{attribute wpf [Container(Layout.Stack)]}
FUNCTION_BLOCK TcoKeyNormalService EXTENDS TcoElements.TcoDi IMPLEMENTS ITcoKeyNormalSevice

VAR

	
	{attribute addProperty Name "<#Key state#> - <#Service#>"}
	_isKeyInService           : BOOL; 

	{attribute addProperty Name "<#Key state#> - <#Normal#>"}
	_isKeyInNormal            : BOOL; 
END_VAR

SUPER^(inoSignal:= inoSignal);


THIS^._isKeyInNormal :=NOT THIS^._signal ;
THIS^._isKeyInService := NOT THIS^._isKeyInNormal;

PROPERTY KeyInNormal : BOOL
GET
KeyInNormal := _isKeyInNormal;
END_GET
END_PROPERTY

PROPERTY KeyInService : BOOL
GET
KeyInService := _isKeyInService;
END_GET
END_PROPERTY

END_FUNCTION_BLOCK

(* stored: Version 1.1.0.1
   POU TcoKeyNormalService: Id {fd8dbc27-6e45-4e78-8f75-e78a5510e99d}, SpecialFunc None
   Property KeyInNormal: Id {ec1426ec-5fce-4c25-9228-d7d73b4c1d65}
   Get Get: Id {0831bc1d-0f68-4b95-897a-ba02076606ba}
   Property KeyInService: Id {72861a8c-56b8-485f-aadb-9e3f4447a674}
   Get Get: Id {07f6d57f-059a-45ef-bef2-3202005cb8fc} *)
